{attribute 'conditionalshow'}
FUNCTION_BLOCK FB_MBRTUMaster_Messages
VAR_INPUT
	{attribute 'hide'}
	bTerminalConfigured					: BOOL;						//Shows that the terminal is configured 
	{attribute 'hide'}
	bError								: BOOL;						//Error from the RTU Function
	{attribute 'hide'}
	bWarning							: BOOL;						//Warning from the RTU Function
	{attribute 'hide'}
	iWarningCode						: INT;						//Warning Code
	{attribute 'hide'}
	iErrorCode							: INT;						//Error Code		
END_VAR
VAR_OUTPUT
	{attribute 'hide'}
	byErrorWarning						: BYTE;						//Error Warning State
	eMessageMBRTUMaster					: E_Message_MBRTUMaster;	//Message from the RTU Master Function
END_VAR
VAR
END_VAR

//Creator : Kai Ebensperger
//Company : Lynus AG
//Date : 08.07.2021
//Version : 1.0.0.0

//With this Funciton is possible to handel the Error and Warning Codes from the Modbus RTU Master.

//Warnings
IF bWarning AND iWarningCode = 0 THEN 
	eMessageMBRTUMaster := E_Message_MBRTUMaster.eNoConnectionToBackend;
END_IF

//Errors
IF bError AND iErrorCode = 1 THEN
	eMessageMBRTUMaster := E_Message_MBRTUMaster.eTooMuchMBRTUMasters;
ELSIF bError AND iErrorCode = 2 THEN
	eMessageMBRTUMaster := E_Message_MBRTUMaster.eTerminalConfigurationError;
ELSIF bError AND iErrorCode = 3 THEN
	eMessageMBRTUMaster := E_Message_MBRTUMaster.eModbusErrorIllegalFunction;
ELSIF bError AND iErrorCode = 4 THEN
	eMessageMBRTUMaster := E_Message_MBRTUMaster.eModbusErrorIllegalDataAdress;
ELSIF bError AND iErrorCode = 5 THEN
	eMessageMBRTUMaster := E_Message_MBRTUMaster.eModbusErrorIllegalDataValue;
ELSIF bError AND iErrorCode = 6 THEN
	eMessageMBRTUMaster := E_Message_MBRTUMaster.eModbusErrorSlaveDeviceFailure;
ELSIF bError AND iErrorCode = 7 THEN
	eMessageMBRTUMaster := E_Message_MBRTUMaster.eModbusErrorAcknowledge;
ELSIF bError AND iErrorCode = 8 THEN
	eMessageMBRTUMaster := E_Message_MBRTUMaster.eModbusErrorSlaveDeviceBusy;
ELSIF bError AND iErrorCode = 9 THEN
	eMessageMBRTUMaster := E_Message_MBRTUMaster.eModbusErrorNegativeAcknowledge;
ELSIF bError AND iErrorCode = 10 THEN
	eMessageMBRTUMaster := E_Message_MBRTUMaster.eModbusErrorMemoryParity;
ELSIF bError AND iErrorCode = 11 THEN
	eMessageMBRTUMaster := E_Message_MBRTUMaster.eModbusErrorGatewayPathUnavailable;
ELSIF bError AND iErrorCode = 12 THEN
	eMessageMBRTUMaster := E_Message_MBRTUMaster.eModbusErrorGatewayTargetDeviceFailedToRespond;
ELSIF bError AND iErrorCode = 13 THEN
	eMessageMBRTUMaster := E_Message_MBRTUMaster.eModbusErrorCharrecTimeout;
ELSIF bError AND iErrorCode = 14 THEN
	eMessageMBRTUMaster := E_Message_MBRTUMaster.eModbusErrorIllegalDataSize;
ELSIF bError AND iErrorCode = 15 THEN
	eMessageMBRTUMaster := E_Message_MBRTUMaster.eModbusErrorIllegalDeviceAdress;
ELSIF bError AND iErrorCode = 16 THEN
	eMessageMBRTUMaster := E_Message_MBRTUMaster.eModbusErrorIllegalDestinationAdress;
ELSIF bError AND iErrorCode = 17 THEN
	eMessageMBRTUMaster := E_Message_MBRTUMaster.eModbusErrorIllegalDestinationSize;
ELSIF bError AND iErrorCode = 18 THEN
	eMessageMBRTUMaster := E_Message_MBRTUMaster.eModbusErrorNoResponse;
ELSIF bError AND iErrorCode = 19 THEN
	eMessageMBRTUMaster := E_Message_MBRTUMaster.eModbusErrorTxBufferOverrun;
ELSIF bError AND iErrorCode = 20 THEN
	eMessageMBRTUMaster := E_Message_MBRTUMaster.eModbusErrorSendTimeout;
ELSIF bError AND iErrorCode = 21 THEN
	eMessageMBRTUMaster := E_Message_MBRTUMaster.eModbusErrorDataSizeOverrun;
ELSIF bError AND iErrorCode = 22 THEN
	eMessageMBRTUMaster := E_Message_MBRTUMaster.eModbusErrorStringOverrun;
ELSIF bError AND iErrorCode = 23 THEN
	eMessageMBRTUMaster := E_Message_MBRTUMaster.eModbusErrorInvalidPointer;
ELSIF bError AND iErrorCode = 24 THEN
	eMessageMBRTUMaster := E_Message_MBRTUMaster.eModbusErrorCRC;
ELSIF bError AND iErrorCode = 25 THEN
	eMessageMBRTUMaster := E_Message_MBRTUMaster.eModbusErrorInvalidMemoryAdress;
ELSIF bError AND iErrorCode = 26 THEN
	eMessageMBRTUMaster := E_Message_MBRTUMaster.eModbusErrorTransmitBufferTooSmal;
END_IF 

IF bWarning THEN 
	byErrorWarning := 1;
END_IF	
	IF bError THEN
		byErrorWarning := 2;
	END_IF

//All ok
IF NOT bError AND NOT bWarning THEN
	eMessageMBRTUMaster := E_Message_MBRTUMaster.eAllOk;
		byErrorWarning := 0;
END_IF

//No Configuration
IF NOT bError AND NOT bTerminalConfigured THEN
	eMessageMBRTUMaster := E_Message_MBRTUMaster.eNoTerminalConfiguration;
END_IF

END_FUNCTION_BLOCK

(* stored: Version 1.1.0.1, ProductVersion 3.1.4024.9
   POU FB_MBRTUMaster_Messages: Id {1edae247-b251-4a9a-9c86-8c4fe43d573a}, SpecialFunc None *)
